FUNCTION_BLOCK CU00xTestMultiPositions EXTENDS TcoDrivesBeckhoff.TcoMultiAxisPositionsRootContainer
VAR_INPUT
END_VAR
VAR_OUTPUT
END_VAR
VAR
	{attribute addProperty Name "<#Pick Position#>"}
	PickPosition:TcoDrivesBeckhoff.TcoMultiAxisMoveParam;
	{attribute addProperty Name "<#Place  Position#>"}
	PlacePosition:TcoDrivesBeckhoff.TcoMultiAxisMoveParam;

END_VAR

PROPERTY PUBLIC PickPos : REFERENCE TO TcoDrivesBeckhoff.TcoMultiAxisMoveParam;
GET
PickPos REF=PickPosition;
END_GET
END_PROPERTY

PROPERTY PUBLIC PlacePos : REFERENCE TO TcoDrivesBeckhoff.TcoMultiAxisMoveParam;
GET
PlacePos REF=PlacePosition;
END_GET
END_PROPERTY

END_FUNCTION_BLOCK

(* stored: Version 1.1.0.1
   POU CU00xTestMultiPositions: Id {cd7dbda4-d274-4cdf-b1b2-8d207511c762}, SpecialFunc None
   Property PickPos: Id {d5f22fa6-de95-492c-a977-aa26e0a454b8}
   Get Get: Id {1bf33f6e-5e82-4ef2-b34c-6b3b63ac4f06}
   Property PlacePos: Id {07ab9d01-eeaf-4668-b9bb-2b28cd21fa1c}
   Get Get: Id {1ef2bda8-305a-4c84-8cae-d55120fc8fd6} *)
